(* PLC project LadderFixture, greenforge-labs codescribe-fixture 1 *)
(* stored: creationDateTime 2020-01-01T00:00:00 *)

PROGRAM Motor_Control
  VAR
    Start_PB : BOOL;
    Stop_PB : BOOL;
    Motor_Run : BOOL := FALSE;
    Fault_In : BOOL;
    Fault_Latch : BOOL;
    Reset_PB : BOOL;
    Ack : BOOL;
    Run_Time : TON;
  END_VAR
  VAR  (* added by the conversion: wires and edge detectors of the diagram *)
    R_TRIG1 : R_TRIG;
  END_VAR

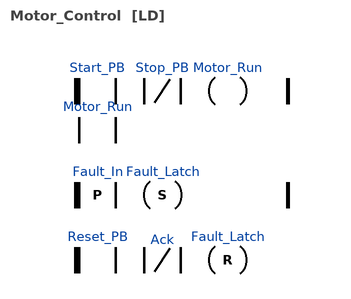
(* LD diagram, written out as Structured Text *)
Motor_Run := (Start_PB OR Motor_Run) AND NOT Stop_PB;
R_TRIG1(CLK := Fault_In);
IF R_TRIG1.Q THEN Fault_Latch := TRUE; END_IF;
IF Reset_PB AND NOT Ack THEN Fault_Latch := FALSE; END_IF;
END_PROGRAM
